TYPE EL2044_Data :
STRUCT
	{attribute addProperty Name "DIG Diag Inputs"}
	_diag : EL2044_Diag;
	{attribute addProperty Name "DIG Inputs Device"}
	_inputs : stDIGInputsDevice;
	{attribute addProperty Name "DIG Outputs"}
	_outputs : EL2044_Outputs;
END_STRUCT
END_TYPE

(* stored: Version 1.1.0.1, ProductVersion 3.1.4024.9
   DUT EL2044_Data: Id {5be5a840-2895-08f5-2743-b1d93b4f432e} *)
